FUNCTION_BLOCK Interval (* Template for an empty simple function block *)
  (* Standard: 61499-1 *)
  (* Version 1.0, 2024-07-26, david *)
  {SET_ATTRIBUTE(OpcUa, DEVICE.SENSOR)}
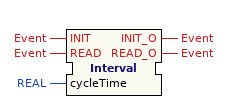
  EVENT_INPUT
    INIT;
    READ;
  END_EVENT
  EVENT_OUTPUT
    INIT_O;
    READ_O;
  END_EVENT
  VAR_INPUT
    cycleTime : REAL; (* Event repetition interval *)
  END_VAR
END_FUNCTION_BLOCK
